// TIA Portal V18 export
DATA_BLOCK "AHUFrostProt"   // DB109
{ S7_Optimized_Access := 'FALSE' }
VERSION : 0.1
// stored: AutoNumber false, DBAccessibleFromOPCUA true, IsOnlyStoredInLoadMemory false, IsWriteProtectedInAS false
   VAR RETAIN
      FrostProt { S7_SetPoint := 'True'} : "UDT_FrostProtection";
   END_VAR
BEGIN
   FrostProt.OATtoStartPreheating[1..3] := 10.0;
END_DATA_BLOCK
